(* PLC project simplified_IXL.project, CODESYS CODESYS V3.5 SP20 *)
(* stored: creationDateTime 2025-01-03T23:08:13.7830976, modificationDateTime 2025-01-03T23:07:12.3834237 *)

{attribute 'qualified_only'}
{attribute 'strict'}
TYPE TC : (TC_101, TC_102, TC_103, TC_104, TC_105, TC_106, TC_107, TC_108, TC_109, TC_110, TC_111, TC_112, TC_113, TC_114, TC_115, TC_116, NIL);
END_TYPE

{attribute 'qualified_only'}
{attribute 'strict'}
TYPE SWITCH : (Sw_01, Sw_02, NIL);
END_TYPE

{attribute 'qualified_only'}
{attribute 'strict'}
TYPE SIGNAL : (Sig_201, Sig_203, Sig_205, Sig_206, Sig_208, NIL);
END_TYPE

TYPE TRAIN_STATE : STRUCT
  exists : BOOL;
  rear_pos : TC;
  front_pos : TC;
  orientation : DIR;
END_STRUCT;
END_TYPE

{attribute 'qualified_only'}
{attribute 'strict'}
TYPE DIR : (DOWN, UP, NIL);
END_TYPE

{attribute 'qualified_only'}
{attribute 'strict'}
TYPE SW_POS : (LEFT, RIGHT, INTERMEDIATE, NIL);
END_TYPE

PROGRAM PLC_PRG
  VAR
    route_state_AB : route_state;
    route_state_BC : route_state;
    route_state_ED : route_state;
    route_state_CD : route_state;
    route_state_DC : route_state;
    route_state_CB : route_state;
    Approaching_train_AB : Approaching_train;
    Approaching_train_BC : Approaching_train;
    Approaching_train_ED : Approaching_train;
    Approaching_train_CD : Approaching_train;
    AUTO_DESTRUCT_AB : AUTO_DESTRUCT;
    AUTO_DESTRUCT_BC : AUTO_DESTRUCT;
    AUTO_DESTRUCT_ED : AUTO_DESTRUCT;
    AUTO_DESTRUCT_CD : AUTO_DESTRUCT;
    AUTO_DESTRUCT_DC : AUTO_DESTRUCT;
    Approaching_train_DC : Approaching_train;
    AUTO_DESTRUCT_CB : AUTO_DESTRUCT;
    Approaching_train_CB : Approaching_train;
  END_VAR
  VAR CONSTANT
    DELAY_DEST_DC : TIME := TIME#30s0ms;
    DELAY_DEST_CB : TIME := TIME#30s0ms;
    DELAY_DEST_ED : TIME := TIME#30s0ms;
    DELAY_DEST_CD : TIME := TIME#30s0ms;
    DELAY_DEST_BC : TIME := TIME#30s0ms;
    DELAY_DEST_AB : TIME := TIME#30s0ms;
  END_VAR
  VAR  (* added by the conversion: wires and edge detectors of the diagram *)
    _AND70000000012_OUT : BOOL;
    _AND80000000011_OUT : BOOL;
  END_VAR

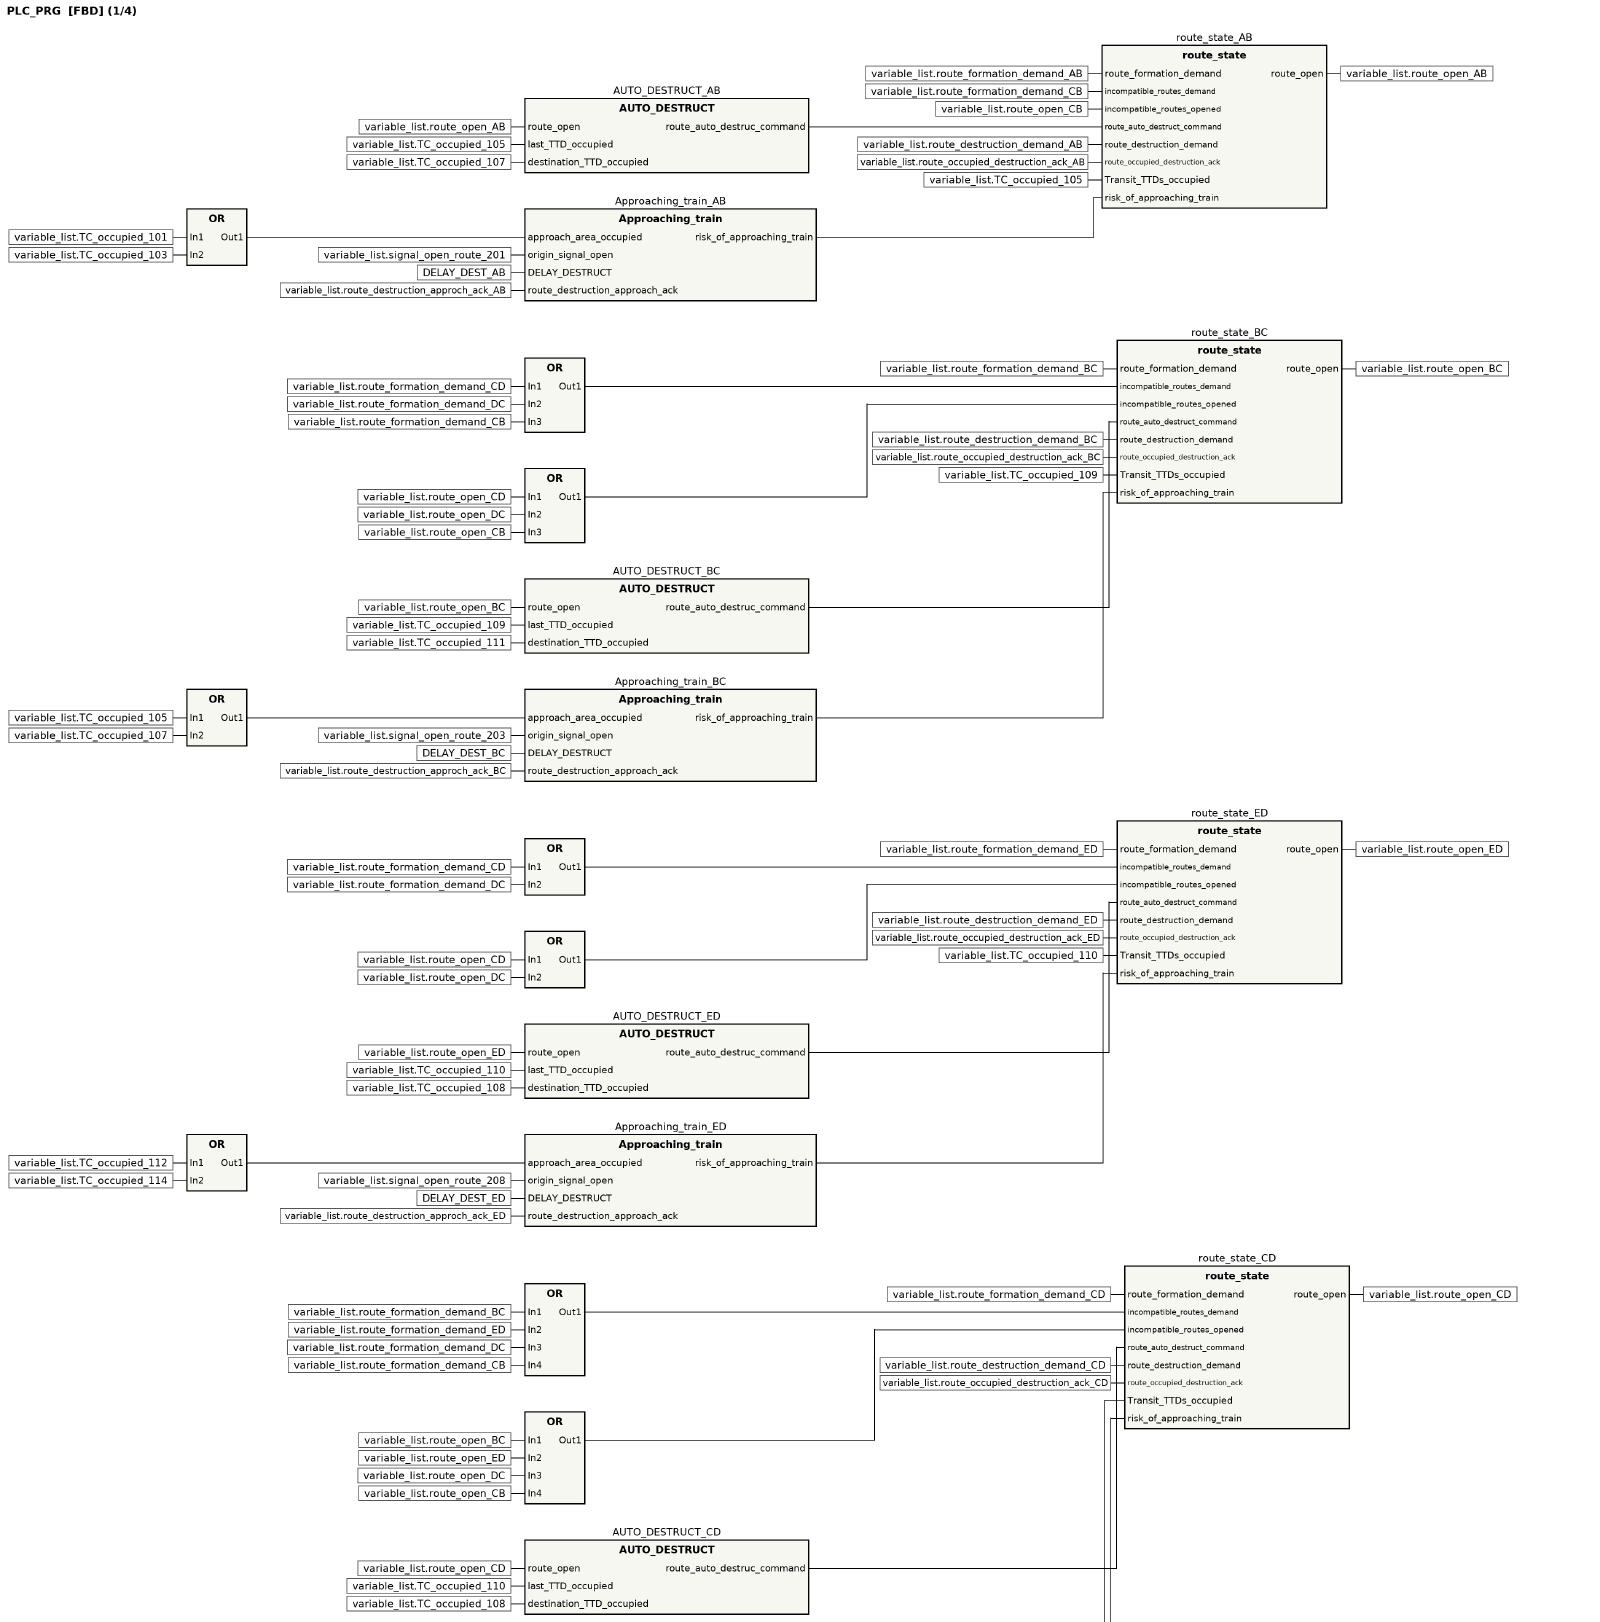
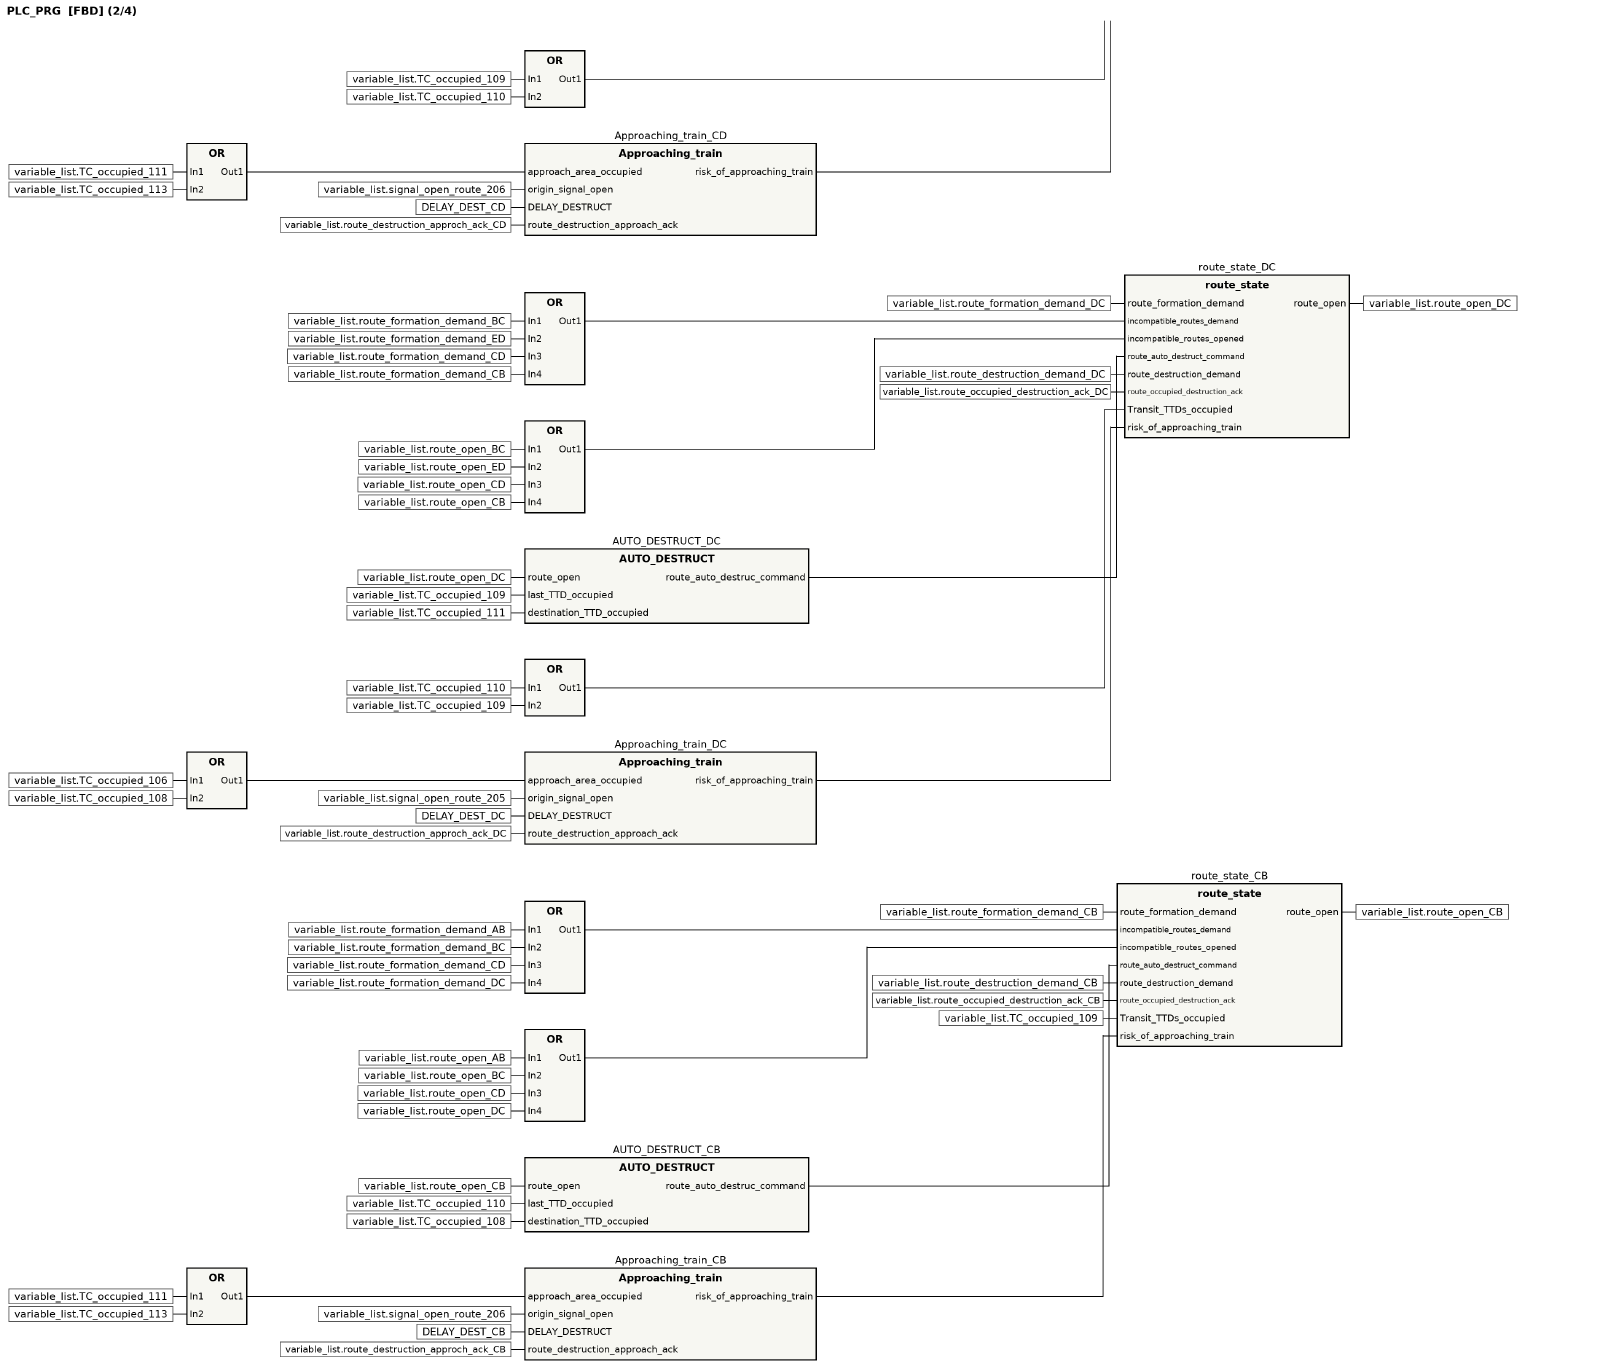
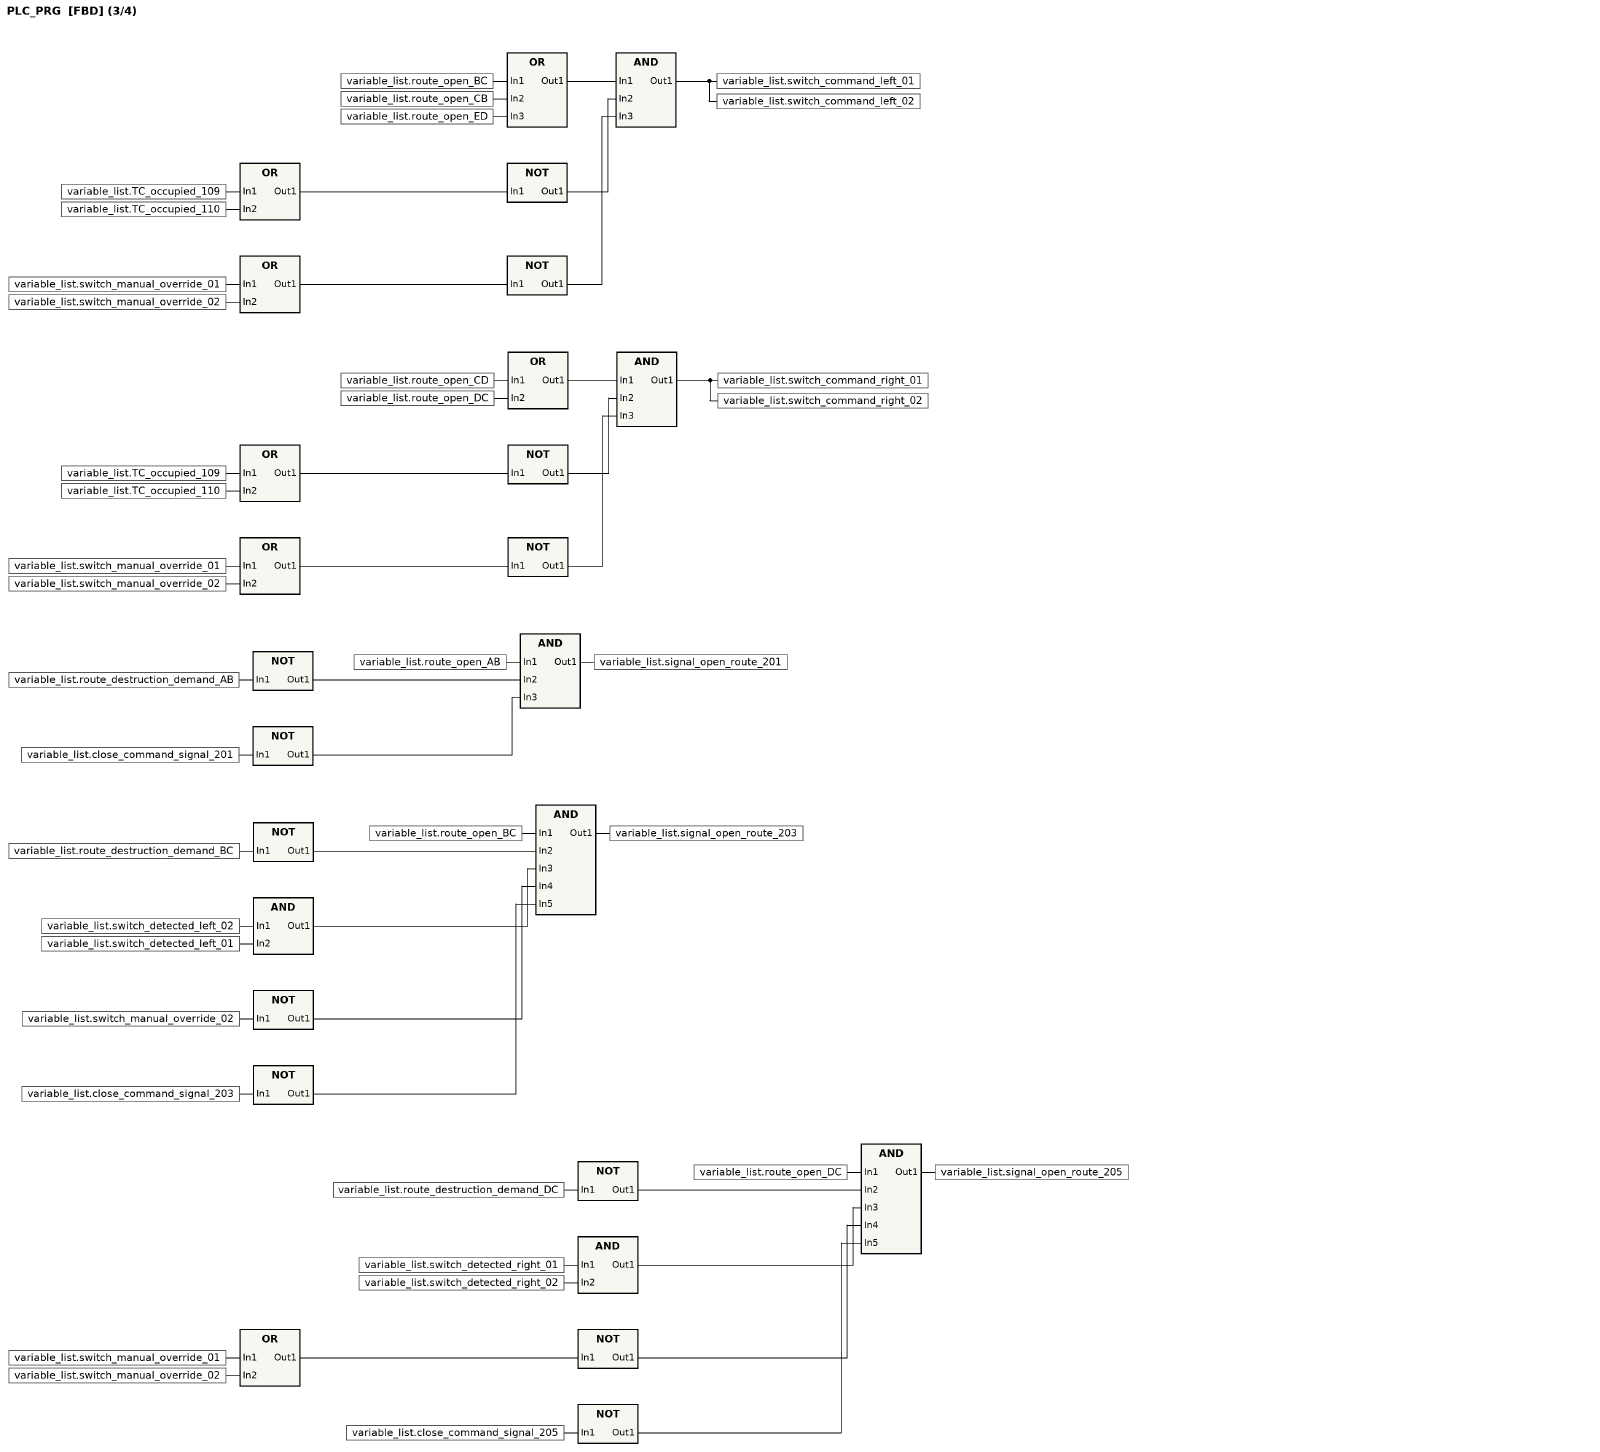
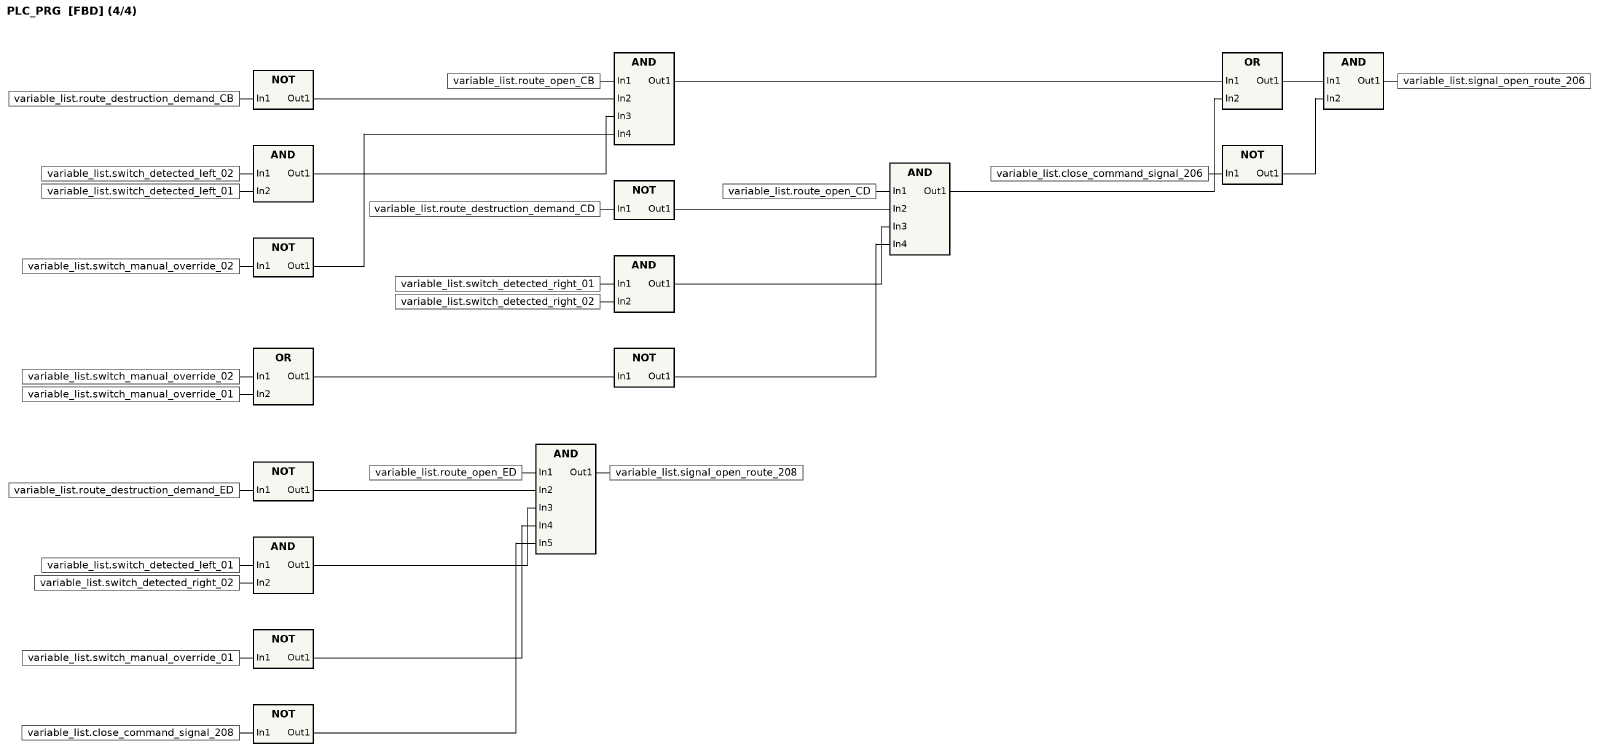
(* FBD diagram, written out as Structured Text *)
AUTO_DESTRUCT_AB(route_open := variable_list.route_open_AB, last_TTD_occupied := variable_list.TC_occupied_105, destination_TTD_occupied := variable_list.TC_occupied_107);
Approaching_train_AB(approach_area_occupied := variable_list.TC_occupied_101 OR variable_list.TC_occupied_103, origin_signal_open := variable_list.signal_open_route_201, DELAY_DESTRUCT := DELAY_DEST_AB, route_destruction_approach_ack := variable_list.route_destruction_approch_ack_AB);
route_state_AB(route_formation_demand := variable_list.route_formation_demand_AB, incompatible_routes_demand := variable_list.route_formation_demand_CB, incompatible_routes_opened := variable_list.route_open_CB, route_auto_destruct_command := AUTO_DESTRUCT_AB.route_auto_destruc_command, route_destruction_demand := variable_list.route_destruction_demand_AB, route_occupied_destruction_ack := variable_list.route_occupied_destruction_ack_AB, Transit_TTDs_occupied := variable_list.TC_occupied_105, risk_of_approaching_train := Approaching_train_AB.risk_of_approaching_train);
variable_list.route_open_AB := route_state_AB.route_open;
AUTO_DESTRUCT_BC(route_open := variable_list.route_open_BC, last_TTD_occupied := variable_list.TC_occupied_109, destination_TTD_occupied := variable_list.TC_occupied_111);
Approaching_train_BC(approach_area_occupied := variable_list.TC_occupied_105 OR variable_list.TC_occupied_107, origin_signal_open := variable_list.signal_open_route_203, DELAY_DESTRUCT := DELAY_DEST_BC, route_destruction_approach_ack := variable_list.route_destruction_approch_ack_BC);
route_state_BC(route_formation_demand := variable_list.route_formation_demand_BC, incompatible_routes_demand := variable_list.route_formation_demand_CD OR variable_list.route_formation_demand_DC OR variable_list.route_formation_demand_CB, incompatible_routes_opened := variable_list.route_open_CD OR variable_list.route_open_DC OR variable_list.route_open_CB, route_auto_destruct_command := AUTO_DESTRUCT_BC.route_auto_destruc_command, route_destruction_demand := variable_list.route_destruction_demand_BC, route_occupied_destruction_ack := variable_list.route_occupied_destruction_ack_BC, Transit_TTDs_occupied := variable_list.TC_occupied_109, risk_of_approaching_train := Approaching_train_BC.risk_of_approaching_train);
variable_list.route_open_BC := route_state_BC.route_open;
AUTO_DESTRUCT_ED(route_open := variable_list.route_open_ED, last_TTD_occupied := variable_list.TC_occupied_110, destination_TTD_occupied := variable_list.TC_occupied_108);
Approaching_train_ED(approach_area_occupied := variable_list.TC_occupied_112 OR variable_list.TC_occupied_114, origin_signal_open := variable_list.signal_open_route_208, DELAY_DESTRUCT := DELAY_DEST_ED, route_destruction_approach_ack := variable_list.route_destruction_approch_ack_ED);
route_state_ED(route_formation_demand := variable_list.route_formation_demand_ED, incompatible_routes_demand := variable_list.route_formation_demand_CD OR variable_list.route_formation_demand_DC, incompatible_routes_opened := variable_list.route_open_CD OR variable_list.route_open_DC, route_auto_destruct_command := AUTO_DESTRUCT_ED.route_auto_destruc_command, route_destruction_demand := variable_list.route_destruction_demand_ED, route_occupied_destruction_ack := variable_list.route_occupied_destruction_ack_ED, Transit_TTDs_occupied := variable_list.TC_occupied_110, risk_of_approaching_train := Approaching_train_ED.risk_of_approaching_train);
variable_list.route_open_ED := route_state_ED.route_open;
AUTO_DESTRUCT_CD(route_open := variable_list.route_open_CD, last_TTD_occupied := variable_list.TC_occupied_110, destination_TTD_occupied := variable_list.TC_occupied_108);
Approaching_train_CD(approach_area_occupied := variable_list.TC_occupied_111 OR variable_list.TC_occupied_113, origin_signal_open := variable_list.signal_open_route_206, DELAY_DESTRUCT := DELAY_DEST_CD, route_destruction_approach_ack := variable_list.route_destruction_approch_ack_CD);
route_state_CD(route_formation_demand := variable_list.route_formation_demand_CD, incompatible_routes_demand := variable_list.route_formation_demand_BC OR variable_list.route_formation_demand_ED OR variable_list.route_formation_demand_DC OR variable_list.route_formation_demand_CB, incompatible_routes_opened := variable_list.route_open_BC OR variable_list.route_open_ED OR variable_list.route_open_DC OR variable_list.route_open_CB, route_auto_destruct_command := AUTO_DESTRUCT_CD.route_auto_destruc_command, route_destruction_demand := variable_list.route_destruction_demand_CD, route_occupied_destruction_ack := variable_list.route_occupied_destruction_ack_CD, Transit_TTDs_occupied := variable_list.TC_occupied_109 OR variable_list.TC_occupied_110, risk_of_approaching_train := Approaching_train_CD.risk_of_approaching_train);
variable_list.route_open_CD := route_state_CD.route_open;
AUTO_DESTRUCT_DC(route_open := variable_list.route_open_DC, last_TTD_occupied := variable_list.TC_occupied_109, destination_TTD_occupied := variable_list.TC_occupied_111);
Approaching_train_DC(approach_area_occupied := variable_list.TC_occupied_106 OR variable_list.TC_occupied_108, origin_signal_open := variable_list.signal_open_route_205, DELAY_DESTRUCT := DELAY_DEST_DC, route_destruction_approach_ack := variable_list.route_destruction_approch_ack_DC);
route_state_DC(route_formation_demand := variable_list.route_formation_demand_DC, incompatible_routes_demand := variable_list.route_formation_demand_BC OR variable_list.route_formation_demand_ED OR variable_list.route_formation_demand_CD OR variable_list.route_formation_demand_CB, incompatible_routes_opened := variable_list.route_open_BC OR variable_list.route_open_ED OR variable_list.route_open_CD OR variable_list.route_open_CB, route_auto_destruct_command := AUTO_DESTRUCT_DC.route_auto_destruc_command, route_destruction_demand := variable_list.route_destruction_demand_DC, route_occupied_destruction_ack := variable_list.route_occupied_destruction_ack_DC, Transit_TTDs_occupied := variable_list.TC_occupied_110 OR variable_list.TC_occupied_109, risk_of_approaching_train := Approaching_train_DC.risk_of_approaching_train);
variable_list.route_open_DC := route_state_DC.route_open;
AUTO_DESTRUCT_CB(route_open := variable_list.route_open_CB, last_TTD_occupied := variable_list.TC_occupied_110, destination_TTD_occupied := variable_list.TC_occupied_108);
Approaching_train_CB(approach_area_occupied := variable_list.TC_occupied_111 OR variable_list.TC_occupied_113, origin_signal_open := variable_list.signal_open_route_206, DELAY_DESTRUCT := DELAY_DEST_CB, route_destruction_approach_ack := variable_list.route_destruction_approch_ack_CB);
route_state_CB(route_formation_demand := variable_list.route_formation_demand_CB, incompatible_routes_demand := variable_list.route_formation_demand_AB OR variable_list.route_formation_demand_BC OR variable_list.route_formation_demand_CD OR variable_list.route_formation_demand_DC, incompatible_routes_opened := variable_list.route_open_AB OR variable_list.route_open_BC OR variable_list.route_open_CD OR variable_list.route_open_DC, route_auto_destruct_command := AUTO_DESTRUCT_CB.route_auto_destruc_command, route_destruction_demand := variable_list.route_destruction_demand_CB, route_occupied_destruction_ack := variable_list.route_occupied_destruction_ack_CB, Transit_TTDs_occupied := variable_list.TC_occupied_109, risk_of_approaching_train := Approaching_train_CB.risk_of_approaching_train);
variable_list.route_open_CB := route_state_CB.route_open;
_AND70000000012_OUT := (variable_list.route_open_BC OR variable_list.route_open_CB OR variable_list.route_open_ED) AND NOT (variable_list.TC_occupied_109 OR variable_list.TC_occupied_110) AND NOT (variable_list.switch_manual_override_01 OR variable_list.switch_manual_override_02);
variable_list.switch_command_left_01 := _AND70000000012_OUT;
variable_list.switch_command_left_02 := _AND70000000012_OUT;
_AND80000000011_OUT := (variable_list.route_open_CD OR variable_list.route_open_DC) AND NOT (variable_list.TC_occupied_109 OR variable_list.TC_occupied_110) AND NOT (variable_list.switch_manual_override_01 OR variable_list.switch_manual_override_02);
variable_list.switch_command_right_01 := _AND80000000011_OUT;
variable_list.switch_command_right_02 := _AND80000000011_OUT;
variable_list.signal_open_route_201 := variable_list.route_open_AB AND NOT variable_list.route_destruction_demand_AB AND NOT variable_list.close_command_signal_201;
variable_list.signal_open_route_203 := variable_list.route_open_BC AND NOT variable_list.route_destruction_demand_BC AND variable_list.switch_detected_left_02 AND variable_list.switch_detected_left_01 AND NOT variable_list.switch_manual_override_02 AND NOT variable_list.close_command_signal_203;
variable_list.signal_open_route_205 := variable_list.route_open_DC AND NOT variable_list.route_destruction_demand_DC AND variable_list.switch_detected_right_01 AND variable_list.switch_detected_right_02 AND NOT (variable_list.switch_manual_override_01 OR variable_list.switch_manual_override_02) AND NOT variable_list.close_command_signal_205;
variable_list.signal_open_route_206 := (variable_list.route_open_CB AND NOT variable_list.route_destruction_demand_CB AND variable_list.switch_detected_left_02 AND variable_list.switch_detected_left_01 AND NOT variable_list.switch_manual_override_02 OR variable_list.route_open_CD AND NOT variable_list.route_destruction_demand_CD AND variable_list.switch_detected_right_01 AND variable_list.switch_detected_right_02 AND NOT (variable_list.switch_manual_override_02 OR variable_list.switch_manual_override_01)) AND NOT variable_list.close_command_signal_206;
variable_list.signal_open_route_208 := variable_list.route_open_ED AND NOT variable_list.route_destruction_demand_ED AND variable_list.switch_detected_left_01 AND variable_list.switch_detected_right_02 AND NOT variable_list.switch_manual_override_01 AND NOT variable_list.close_command_signal_208;
END_PROGRAM

{attribute 'do_checks_for_implicit_code'}
FUNCTION_BLOCK AUTO_DESTRUCT
  VAR_INPUT
    route_open : BOOL;
    last_TTD_occupied : BOOL;
    destination_TTD_occupied : BOOL;
  END_VAR
  VAR_OUTPUT
    route_auto_destruc_command : BOOL;
  END_VAR

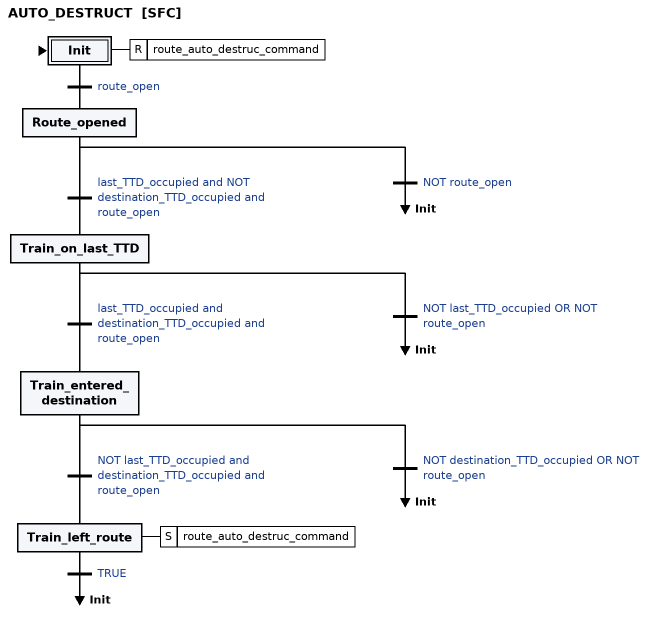
INITIAL_STEP Init:
  route_auto_destruc_command(R);
END_STEP
TRANSITION FROM Init TO Route_opened
  := route_open;
END_TRANSITION
STEP Route_opened:
END_STEP
TRANSITION FROM Route_opened TO Train_on_last_TTD
  := last_TTD_occupied and NOT destination_TTD_occupied and route_open;
END_TRANSITION
TRANSITION FROM Route_opened TO Init
  := NOT route_open;
END_TRANSITION
STEP Train_on_last_TTD:
END_STEP
TRANSITION FROM Train_on_last_TTD TO Train_entered_destination
  := last_TTD_occupied and destination_TTD_occupied and route_open;
END_TRANSITION
TRANSITION FROM Train_on_last_TTD TO Init
  := NOT last_TTD_occupied OR NOT route_open;
END_TRANSITION
STEP Train_entered_destination:
END_STEP
TRANSITION FROM Train_entered_destination TO Train_left_route
  := NOT last_TTD_occupied and destination_TTD_occupied and route_open;
END_TRANSITION
TRANSITION FROM Train_entered_destination TO Init
  := NOT destination_TTD_occupied OR NOT route_open;
END_TRANSITION
STEP Train_left_route:
  route_auto_destruc_command(S);
END_STEP
TRANSITION FROM Train_left_route TO Init
  := TRUE;
END_TRANSITION
END_FUNCTION_BLOCK

FUNCTION_BLOCK route_state
  VAR_INPUT
    route_formation_demand : BOOL;
    incompatible_routes_demand : BOOL;
    incompatible_routes_opened : BOOL;
    route_auto_destruct_command : BOOL;
    route_destruction_demand : BOOL;
    route_occupied_destruction_ack : BOOL;
  END_VAR
  VAR_OUTPUT
    route_open : BOOL;
  END_VAR
  VAR
    SR_route : SR;
    Auto_destruct_state_machine : AUTO_DESTRUCT;
  END_VAR
  VAR_INPUT
    Transit_TTDs_occupied : BOOL;
    risk_of_approaching_train : BOOL;
  END_VAR

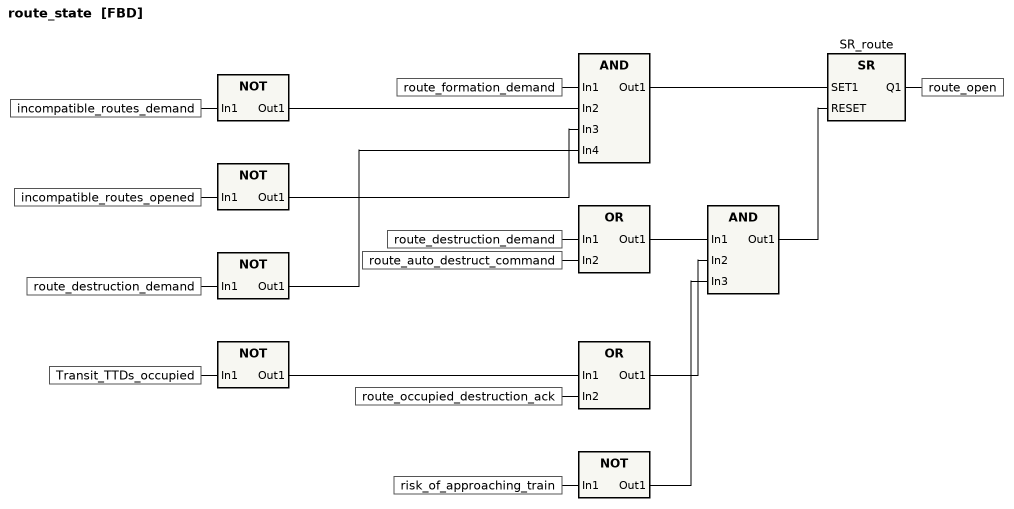
(* FBD diagram, written out as Structured Text *)
SR_route(SET1 := route_formation_demand AND NOT incompatible_routes_demand AND NOT incompatible_routes_opened AND NOT route_destruction_demand, RESET := (route_destruction_demand OR route_auto_destruct_command) AND (NOT Transit_TTDs_occupied OR route_occupied_destruction_ack) AND NOT risk_of_approaching_train);
route_open := SR_route.Q1;
END_FUNCTION_BLOCK

FUNCTION_BLOCK Approaching_train
  VAR_INPUT
    approach_area_occupied : BOOL;
    origin_signal_open : BOOL;
    {attribute 'input_constant'}
    DELAY_DESTRUCT : TIME;
    route_destruction_approach_ack : BOOL;
  END_VAR
  VAR_OUTPUT
    risk_of_approaching_train : BOOL;
  END_VAR
  VAR
    TON_approach_timer : TON;
    SR_approaching_train : SR;
  END_VAR

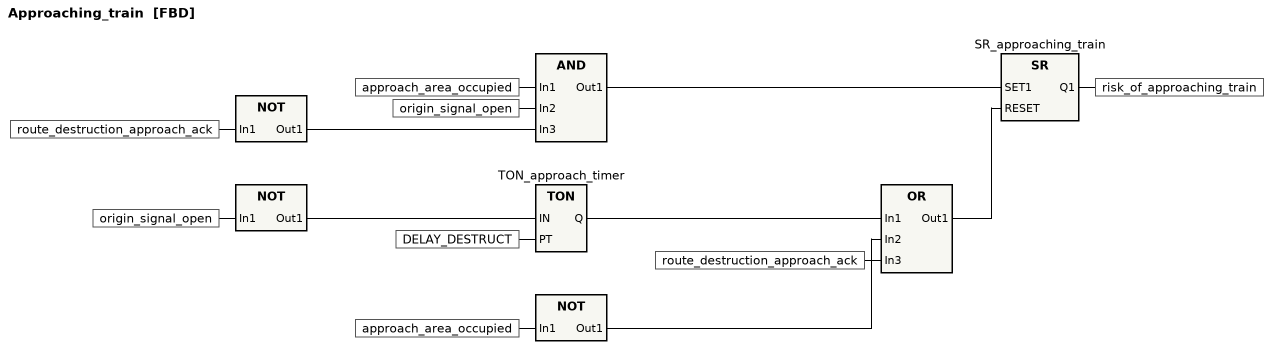
(* FBD diagram, written out as Structured Text *)
TON_approach_timer(IN := NOT origin_signal_open, PT := DELAY_DESTRUCT);
SR_approaching_train(SET1 := approach_area_occupied AND origin_signal_open AND NOT route_destruction_approach_ack, RESET := TON_approach_timer.Q OR NOT approach_area_occupied OR route_destruction_approach_ack);
risk_of_approaching_train := SR_approaching_train.Q1;
END_FUNCTION_BLOCK

PROGRAM simulation
  VAR
    NOT_switch_detected_left_01 : BOOL;
    NOT_switch_detected_right_01 : BOOL;
    NOT_switch_detected_left_02 : BOOL;
    NOT_switch_detected_right_02 : BOOL;
    NOT_switch_middle_01 : BOOL;
    NOT_switch_middle_02 : BOOL;
    switch_commanded_01 : BOOL;
    switch_commanded_02 : BOOL;
    switch_moving_01 : BOOL;
    switch_moving_02 : BOOL;
    Trains : ARRAY[1..6] OF TRAIN_STATE := [6((rear_pos := TC.NIL, front_pos := TC.NIL, orientation := DIR.NIL))];
  END_VAR

                    
NOT_switch_detected_left_01 := NOT(variable_list.switch_detected_left_01);
NOT_switch_detected_left_02 := NOT(variable_list.switch_detected_left_02);
NOT_switch_detected_right_01 := NOT(variable_list.switch_detected_right_01);
NOT_switch_detected_right_02 := NOT(variable_list.switch_detected_right_02);

NOT_switch_middle_01 := variable_list.switch_detected_left_01 OR variable_list.switch_detected_right_01;
NOT_switch_middle_02 := variable_list.switch_detected_left_02 OR variable_list.switch_detected_right_02;

switch_commanded_01 := variable_list.switch_command_left_01 OR variable_list.switch_command_right_01;
switch_commanded_02 := variable_list.switch_command_left_02 OR variable_list.switch_command_right_02;

switch_moving_01 :=
		variable_list.switch_command_left_01 AND NOT(variable_list.switch_detected_left_01) 
	OR	variable_list.switch_command_right_01 AND NOT(variable_list.switch_detected_right_01) ;
switch_moving_02 :=
		variable_list.switch_command_left_02 AND NOT(variable_list.switch_detected_left_02) 
	OR	variable_list.switch_command_right_02 AND NOT(variable_list.switch_detected_right_02) ;


                  
END_PROGRAM

FUNCTION Next_TC : TC
  VAR_INPUT
    tc : TC;
    dir : DIR;
    sw_pos_1 : SW_POS;
    sw_pos_2 : SW_POS;
  END_VAR
  VAR_OUTPUT
    nexttc : TC;
  END_VAR

                    IF dir = DIR.UP THEN
	IF tc = TC.TC_101 THEN
		nexttc := TC.TC_103;
	ELSE IF tc = TC.TC_102 THEN
		nexttc := TC.TC_104;
	ELSE IF tc = TC.TC_103 THEN
		nexttc := TC.TC_105;
	ELSE IF tc = TC.TC_104 THEN
		nexttc := TC.TC_106;
	ELSE IF tc = TC.TC_105 THEN
		nexttc := TC.TC_107;
	ELSE IF tc = TC.TC_106 THEN
		nexttc := TC.TC_108;
	ELSE IF tc = TC.TC_107 THEN
		nexttc := TC.TC_109;
	ELSE IF tc = TC.TC_108 THEN
		nexttc := TC.TC_110;
	ELSE IF tc = TC.TC_109 THEN
		nexttc := TC.TC_111;
	ELSE IF tc = TC.TC_110 THEN
		IF sw_pos_1 = SW_POS.LEFT THEN
			nexttc := TC.TC_112;
		ELSE IF sw_pos_1 = SW_POS.RIGHT THEN
			nexttc := TC.TC_109;
		ELSE (* sw_pos_1 = SW_POS.NIL *)
			nexttc := TC.NIL;
		END_IF END_IF
	ELSE IF tc = TC.TC_111 THEN
		nexttc := TC.TC_113;
	ELSE IF tc = TC.TC_112 THEN
		nexttc := TC.TC_114;
	ELSE IF tc = TC.TC_113 THEN
		nexttc := TC.TC_115;
	ELSE IF tc = TC.TC_114 THEN
		nexttc := TC.TC_116;
	ELSE IF tc = TC.TC_115 THEN
		nexttc := TC.NIL;
	ELSE IF tc = TC.TC_116 THEN
		nexttc := TC.NIL;
	ELSE (* tc = TC.NIL *)
		nexttc := TC.NIL;
	END_IF END_IF END_IF END_IF END_IF END_IF END_IF END_IF END_IF END_IF END_IF END_IF END_IF END_IF END_IF END_IF
	
ELSE IF dir = DIR.DOWN THEN
	IF tc = TC.TC_101 THEN
		nexttc := TC.NIL;
	ELSE IF tc = TC.TC_102 THEN
		nexttc := TC.NIL;
	ELSE IF tc = TC.TC_103 THEN
		nexttc := TC.TC_101;
	ELSE IF tc = TC.TC_104 THEN
		nexttc := TC.TC_102;
	ELSE IF tc = TC.TC_105 THEN
		nexttc := TC.TC_103;
	ELSE IF tc = TC.TC_106 THEN
		nexttc := TC.TC_104;
	ELSE IF tc = TC.TC_107 THEN
		nexttc := TC.TC_105;
	ELSE IF tc = TC.TC_108 THEN
		nexttc := TC.TC_106;
	ELSE IF tc = TC.TC_109 THEN
		IF sw_pos_2 = SW_POS.LEFT THEN
			nexttc := TC.TC_107;
		ELSE IF sw_pos_2 = SW_POS.RIGHT THEN
			nexttc := TC.TC_110;
		ELSE (* sw_pos_2 = SW_POS.NIL *)
			nexttc := TC.NIL;
		END_IF END_IF
	ELSE IF tc = TC.TC_110 THEN
		nexttc := TC.TC_108;
	ELSE IF tc = TC.TC_111 THEN
		nexttc := TC.TC_109;
	ELSE IF tc = TC.TC_112 THEN
		nexttc := TC.TC_110;
	ELSE IF tc = TC.TC_113 THEN
		nexttc := TC.TC_111;
	ELSE IF tc = TC.TC_114 THEN
		nexttc := TC.TC_112;
	ELSE IF tc = TC.TC_115 THEN
		nexttc := TC.TC_113;
	ELSE IF tc = TC.TC_116 THEN
		nexttc := TC.TC_114;
	ELSE (* tc = TC.NIL *)
		nexttc := TC.NIL;
	END_IF END_IF END_IF END_IF END_IF END_IF END_IF END_IF END_IF END_IF END_IF END_IF END_IF END_IF END_IF END_IF

ELSE (* dir = DIR.NIL *)
	nexttc := TC.NIL;
END_IF END_IF
                  
END_FUNCTION

CONFIGURATION Device
  RESOURCE Application ON PLC
    {attribute 'qualified_only'}
    VAR_GLOBAL  (* variable_list *)
      TC_occupied_101 AT %IX0.0 : BOOL := FALSE;
      TC_occupied_103 AT %IX0.1 : BOOL := FALSE;
      TC_occupied_105 AT %IX0.2 : BOOL := FALSE;
      TC_occupied_107 AT %IX0.3 : BOOL := FALSE;
      TC_occupied_109 AT %IX0.4 : BOOL := FALSE;
      TC_occupied_111 AT %IX0.5 : BOOL := FALSE;
      TC_occupied_113 AT %IX0.6 : BOOL := FALSE;
      TC_occupied_115 AT %IX0.7 : BOOL := FALSE;
      TC_occupied_102 AT %IX1.0 : BOOL := FALSE;
      TC_occupied_104 AT %IX1.1 : BOOL := FALSE;
      TC_occupied_106 AT %IX1.2 : BOOL := FALSE;
      TC_occupied_108 AT %IX1.3 : BOOL := FALSE;
      TC_occupied_110 AT %IX1.4 : BOOL := FALSE;
      TC_occupied_112 AT %IX1.5 : BOOL := FALSE;
      TC_occupied_114 AT %IX1.6 : BOOL := FALSE;
      TC_occupied_116 AT %IX1.7 : BOOL := FALSE;
      switch_detected_left_01 : BOOL := FALSE;
      switch_detected_right_01 : BOOL := FALSE;
      switch_detected_left_02 : BOOL := FALSE;
      switch_detected_right_02 : BOOL := FALSE;
      route_destruction_demand_AB : BOOL := FALSE;
      route_destruction_demand_BC : BOOL := FALSE;
      route_destruction_demand_ED : BOOL := FALSE;
      route_destruction_demand_CD : BOOL := FALSE;
      route_destruction_demand_DC : BOOL := FALSE;
      route_destruction_demand_CB : BOOL := FALSE;
      route_formation_demand_AB : BOOL := FALSE;
      route_formation_demand_BC : BOOL := FALSE;
      route_formation_demand_ED : BOOL := FALSE;
      route_formation_demand_CD : BOOL := FALSE;
      route_formation_demand_DC : BOOL := FALSE;
      route_formation_demand_CB : BOOL := FALSE;
      switch_manual_override_01 : BOOL := FALSE;
      switch_manual_override_02 : BOOL := FALSE;
      close_command_signal_201 : BOOL := FALSE;
      close_command_signal_203 : BOOL := FALSE;
      close_command_signal_205 : BOOL := FALSE;
      close_command_signal_206 : BOOL := FALSE;
      close_command_signal_208 : BOOL := FALSE;
      signal_open_route_201 : BOOL := FALSE;
      signal_open_route_203 : BOOL := FALSE;
      signal_open_route_205 : BOOL := FALSE;
      signal_open_route_206 : BOOL := FALSE;
      signal_open_route_208 : BOOL := FALSE;
      switch_command_left_01 : BOOL := FALSE;
      switch_command_right_01 : BOOL := FALSE;
      switch_command_left_02 : BOOL := FALSE;
      switch_command_right_02 : BOOL := FALSE;
      route_open_AB : BOOL := FALSE;
      route_open_BC : BOOL := FALSE;
      route_open_ED : BOOL := FALSE;
      route_open_CD : BOOL := FALSE;
      route_open_DC : BOOL := FALSE;
      route_open_CB : BOOL := FALSE;
      route_occupied_destruction_ack_AB : BOOL := FALSE;
      route_occupied_destruction_ack_BC : BOOL := FALSE;
      route_occupied_destruction_ack_ED : BOOL := FALSE;
      route_occupied_destruction_ack_CD : BOOL := FALSE;
      route_occupied_destruction_ack_DC : BOOL := FALSE;
      route_occupied_destruction_ack_CB : BOOL := FALSE;
      route_destruction_approch_ack_AB : BOOL := FALSE;
      route_destruction_approch_ack_BC : BOOL := FALSE;
      route_destruction_approch_ack_ED : BOOL := FALSE;
      route_destruction_approch_ack_CD : BOOL := FALSE;
      route_destruction_approch_ack_DC : BOOL := FALSE;
      route_destruction_approch_ack_CB : BOOL := FALSE;
    END_VAR
    TASK MainTask(INTERVAL := T#20ms, PRIORITY := 1);
    TASK VISU_TASK(INTERVAL := T#100ms, PRIORITY := 31);
    PROGRAM PLC_PRG WITH MainTask : PLC_PRG;
    PROGRAM simulation WITH MainTask : simulation;
    PROGRAM VisuElems.Visu_Prg WITH VISU_TASK : VisuElems.Visu_Prg;
  END_RESOURCE
END_CONFIGURATION
